{attribute 'linkalways'} 
{attribute 'no_explicit_call' := 'This FB is a CLASS and must be accessed using methods or properties'}
{attribute 'enable_dynamic_creation'}
FUNCTION_BLOCK Node_F_VN_GradeDataMatrixCode EXTENDS VisionNode
VAR
    ipSrcImage : _ITcVnImage;
    ipDecodedData : _ITcVnContainer;
    stCodeGrades : 	_TcVnCodeGradesDM;
    fModuleWidth : _REAL(4.0);
    fAngleDeg : _REAL(0.0);
    hrPrev : _HRESULT(S_OK);
	hresult : _HRESULT(S_OK);
END_VAR

METHOD PUBLIC  Clone : I_Node
VAR
	pNode : POINTER TO Node_F_VN_GradeDataMatrixCode;
END_VAR
pNode := __NEW(Node_F_VN_GradeDataMatrixCode);
Clone := pNode^;
END_METHOD

METHOD FB_init : BOOL
VAR_INPUT
	bInitRetains : BOOL; // if TRUE, the retain variables are initialized (warm start / cold start)
	bInCopyCode : BOOL;  // if TRUE, the instance afterwards gets moved into the copy code (online change)
END_VAR
AddInput('ipSrcImage', ipSrcImage);
AddParameter('fModuleWidth', fModuleWidth);
AddInput('hrPrev', hrPrev);
AddOutput('ipDecodedData', ipDecodedData);
AddOutput('stCodeGrades', stCodeGrades);
AddOutput('fAngleDeg', fAngleDeg);
AddOutput('hresult', hresult);
END_METHOD

METHOD PROTECTED OnExecute
VAR
    angle : REAL;
END_VAR
hresult.Value := F_VN_GradeDataMatrixCode(
	ipSrcImage := ipSrcImage.Value,
    ipDecodedData := ipDecodedData.Value,
    stCodeGrades := stCodeGrades.Value,
    fModuleWidth := fModuleWidth.Value,
	hrPrev:= hrPrev.Value,
    fAngleDeg => angle);

fAngleDeg.Value := angle;
END_METHOD

METHOD PUBLIC PreExecutionCheck
VAR_INPUT
	Check : I_PreExecutionChecks;
END_VAR
Check.IsTrue(ipSrcImage.IsValid, 'ipSrcImage must contain an image');
Check.IsTrue(ipSrcImage.HasChannelCount(1), 'ipSrcImage must have 1 channel');
Check.IsTrue(ipSrcImage.IsPixelDepth(8), 'ipSrcImage must have 8 bit pixel depth');
Check.IsTrue(fModuleWidth.Value >= 3, 'fModuleWidth must be greater than or equal to 3');
END_METHOD

END_FUNCTION_BLOCK

(* stored: Version 1.1.0.1, ProductVersion 3.1.4024.13
   POU Node_F_VN_GradeDataMatrixCode: Id {3170efb5-b900-037d-0c62-0af9849fc066}, SpecialFunc None
   Folder Constructor: Id {c21b6b0c-df48-04c4-0b76-862d463fef18}
   Method Clone: Id {1243dccc-3374-0c6b-16a2-6cfc6ec66fd5}
   Method FB_init: Id {2382fc58-511b-0f49-0025-c04023342627}
   Method OnExecute: Id {1107cd5b-ce12-0d93-00c8-cc15c0109bed}
   Method PreExecutionCheck: Id {0ccee4eb-d2c3-0904-1999-61eb2bcc9d9e} *)
